// TIA Portal V21 export
DATA_BLOCK "MotorPump"   // DB2
{ S7_Optimized_Access := 'TRUE' }
// stored: MemoryReserve 100
   VAR
      Motor1 : Array[0..5] of "Motor_template";
   END_VAR
BEGIN
END_DATA_BLOCK
